Staubli VAL3: buildList.pgx

program buildList()
  local num l_nSize
  local string l_sEvent
  local num i
  local string l_sEmpty
begin
  // INIT the list
  l_sEmpty=""
  call use:stringCopy(l_sEmpty,sList)
  // Build the list
  for i=0 to size(saveData:fFrameItem)-1
    call listAdd(toString("2",i)+" "+saveData:fFrameItem[i].sName)
  endFor
end
